// TIA Portal V20 program export: 0 tag tables, 0 data types, 0 data blocks, 3 code blocks (in call order from the OBs), 1 instance data blocks

ORGANIZATION_BLOCK "Main"   // OB1, LAD, ProgramCycle
TITLE = "Main Program Sweep (Cycle)"
{ S7_Optimized_Access := 'TRUE' }
// stored: SetENOAutomatically false
   VAR_INPUT
      Initial_Call : Bool;   // Initial call of this OB
      Remanence : Bool;   // =True, if remanent data are available
   END_VAR
   VAR_TEMP
      tst : Bool;
      tst_ergebnis : Bool;
   END_VAR
BEGIN

REGION Network 1: Testchange
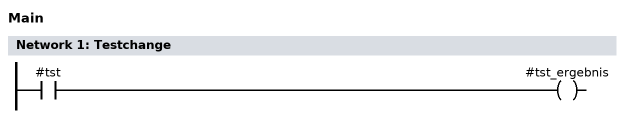
   RUNG wire#powerrail
      Contact( #tst )
      Coil( #tst_ergebnis )
   END_RUNG
   // the same network as SCL:
   #tst_ergebnis := #tst;
END_REGION
END_ORGANIZATION_BLOCK

FUNCTION_BLOCK "Main_Safety_RTG1"   // FB1, F_FBD
{ S7_Optimized_Access := 'TRUE' }
// stored: AutoNumber false
BEGIN
END_FUNCTION_BLOCK

FUNCTION_BLOCK "Block_1"
{ S7_Optimized_Access := 'TRUE' }
VERSION : 0.1
   VAR_INPUT 
      i_test : Bool;
   END_VAR

   VAR_OUTPUT 
      o_test : Bool;
   END_VAR


BEGIN
	// Comment for test
	IF #i_test THEN
	    #o_test := true;
	ELSE
	    #o_test := false;
	END_IF;
	
	//Popel
	//asdf
END_FUNCTION_BLOCK

DATA_BLOCK "Main_Safety_RTG1_DB"   // DB1, F_DB
NAME : FUSI
// stored: InstanceOfName Main_Safety_RTG1, InstanceOfType FB
"Main_Safety_RTG1"
BEGIN
END_DATA_BLOCK
